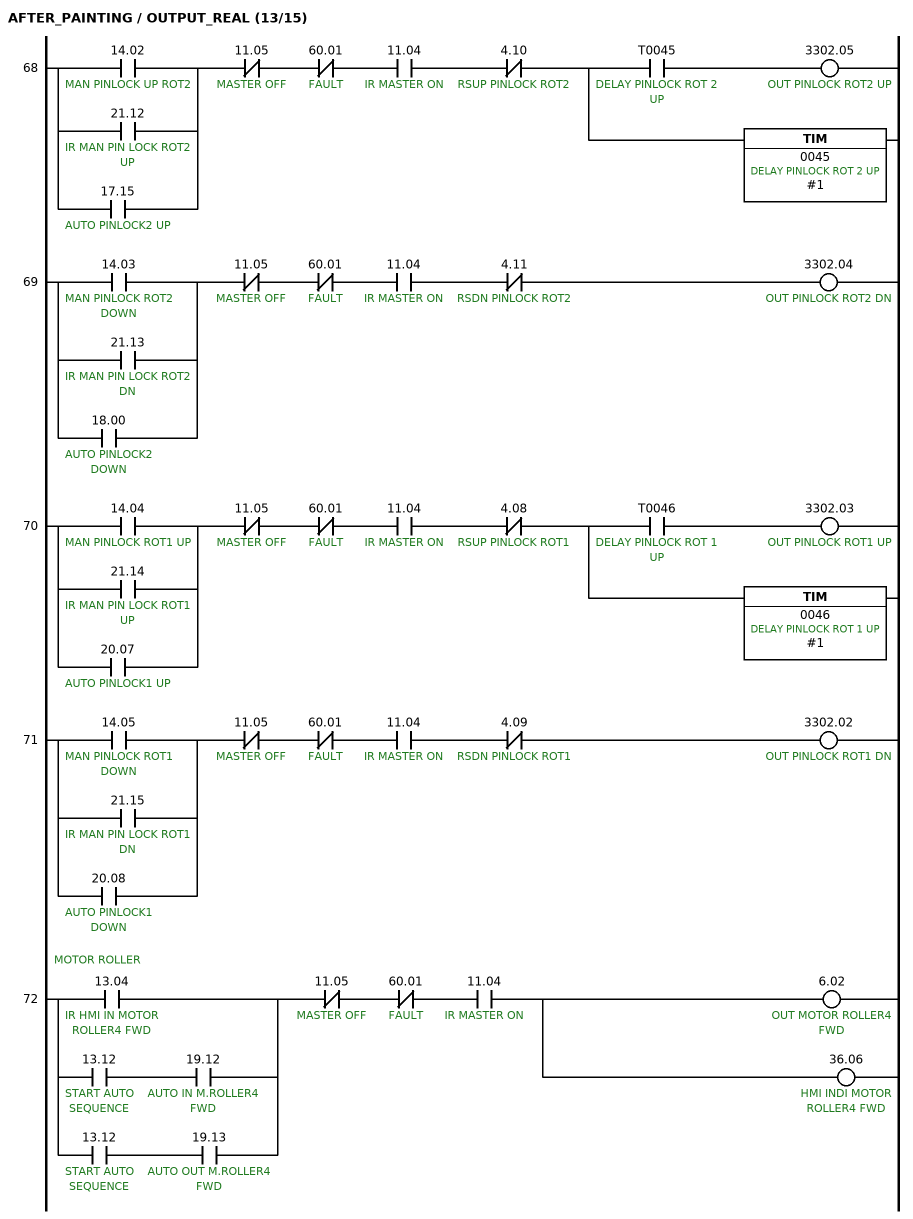
; [picture p24: AFTER_PAINTING / OUTPUT_REAL, rungs 68-72]
; rung 68
LD 14.02  ; MAN PINLOCK UP ROT2
OR 21.12  ; IR MAN PIN LOCK ROT2 UP
OR 17.15  ; AUTO PINLOCK2 UP
ANDNOT 11.05  ; MASTER OFF
ANDNOT 60.01  ; FAULT
AND 11.04  ; IR MASTER ON
ANDNOT 4.10  ; RSUP PINLOCK ROT2
OUT TR0
AND T0045  ; DELAY PINLOCK ROT 2 UP
OUT 3302.05  ; OUT PINLOCK ROT2 UP
LD TR0
TIM 0045 #1  ; DELAY PINLOCK ROT 2 UP
; rung 69
LD 14.03  ; MAN PINLOCK ROT2 DOWN
OR 21.13  ; IR MAN PIN LOCK ROT2 DN
OR 18.00  ; AUTO PINLOCK2 DOWN
ANDNOT 11.05  ; MASTER OFF
ANDNOT 60.01  ; FAULT
AND 11.04  ; IR MASTER ON
ANDNOT 4.11  ; RSDN PINLOCK ROT2
OUT 3302.04  ; OUT PINLOCK ROT2 DN
; rung 70
LD 14.04  ; MAN PINLOCK ROT1 UP
OR 21.14  ; IR MAN PIN LOCK ROT1 UP
OR 20.07  ; AUTO PINLOCK1 UP
ANDNOT 11.05  ; MASTER OFF
ANDNOT 60.01  ; FAULT
AND 11.04  ; IR MASTER ON
ANDNOT 4.08  ; RSUP PINLOCK ROT1
OUT TR0
AND T0046  ; DELAY PINLOCK ROT 1 UP
OUT 3302.03  ; OUT PINLOCK ROT1 UP
LD TR0
TIM 0046 #1  ; DELAY PINLOCK ROT 1 UP
; rung 71
LD 14.05  ; MAN PINLOCK ROT1 DOWN
OR 21.15  ; IR MAN PIN LOCK ROT1 DN
OR 20.08  ; AUTO PINLOCK1 DOWN
ANDNOT 11.05  ; MASTER OFF
ANDNOT 60.01  ; FAULT
AND 11.04  ; IR MASTER ON
ANDNOT 4.09  ; RSDN PINLOCK ROT1
OUT 3302.02  ; OUT PINLOCK ROT1 DN
; rung 72: MOTOR ROLLER
LD 13.04  ; IR HMI IN MOTOR ROLLER4 FWD
LD 13.12  ; START AUTO SEQUENCE
AND 19.12  ; AUTO IN M.ROLLER4 FWD
ORLD
LD 13.12  ; START AUTO SEQUENCE
AND 19.13  ; AUTO OUT M.ROLLER4 FWD
ORLD
ANDNOT 11.05  ; MASTER OFF
ANDNOT 60.01  ; FAULT
AND 11.04  ; IR MASTER ON
OUT 6.02  ; OUT MOTOR ROLLER4 FWD
OUT 36.06  ; HMI INDI MOTOR ROLLER4 FWD

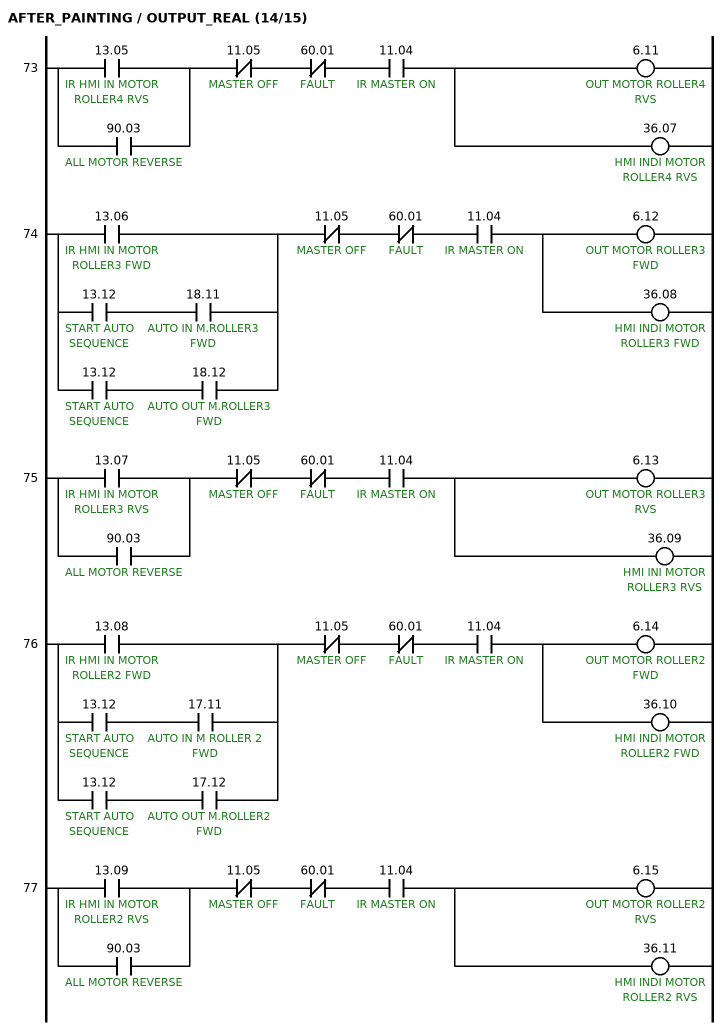
; rung 73
LD 13.05  ; IR HMI IN MOTOR ROLLER4 RVS
OR 90.03  ; ALL MOTOR REVERSE
ANDNOT 11.05  ; MASTER OFF
ANDNOT 60.01  ; FAULT
AND 11.04  ; IR MASTER ON
OUT 6.11  ; OUT MOTOR ROLLER4 RVS
OUT 36.07  ; HMI INDI MOTOR ROLLER4 RVS
; rung 74
LD 13.06  ; IR HMI IN MOTOR ROLLER3 FWD
LD 13.12  ; START AUTO SEQUENCE
AND 18.11  ; AUTO IN M.ROLLER3 FWD
ORLD
LD 13.12  ; START AUTO SEQUENCE
AND 18.12  ; AUTO OUT M.ROLLER3 FWD
ORLD
ANDNOT 11.05  ; MASTER OFF
ANDNOT 60.01  ; FAULT
AND 11.04  ; IR MASTER ON
OUT 6.12  ; OUT MOTOR ROLLER3 FWD
OUT 36.08  ; HMI INDI MOTOR ROLLER3 FWD
; rung 75
LD 13.07  ; IR HMI IN MOTOR ROLLER3 RVS
OR 90.03  ; ALL MOTOR REVERSE
ANDNOT 11.05  ; MASTER OFF
ANDNOT 60.01  ; FAULT
AND 11.04  ; IR MASTER ON
OUT 6.13  ; OUT MOTOR ROLLER3 RVS
OUT 36.09  ; HMI INI MOTOR ROLLER3 RVS
; rung 76
LD 13.08  ; IR HMI IN MOTOR ROLLER2 FWD
LD 13.12  ; START AUTO SEQUENCE
AND 17.11  ; AUTO IN M ROLLER 2 FWD
ORLD
LD 13.12  ; START AUTO SEQUENCE
AND 17.12  ; AUTO OUT M.ROLLER2 FWD
ORLD
ANDNOT 11.05  ; MASTER OFF
ANDNOT 60.01  ; FAULT
AND 11.04  ; IR MASTER ON
OUT 6.14  ; OUT MOTOR ROLLER2 FWD
OUT 36.10  ; HMI INDI MOTOR ROLLER2 FWD
; rung 77
LD 13.09  ; IR HMI IN MOTOR ROLLER2 RVS
OR 90.03  ; ALL MOTOR REVERSE
ANDNOT 11.05  ; MASTER OFF
ANDNOT 60.01  ; FAULT
AND 11.04  ; IR MASTER ON
OUT 6.15  ; OUT MOTOR ROLLER2 RVS
OUT 36.11  ; HMI INDI MOTOR ROLLER2 RVS

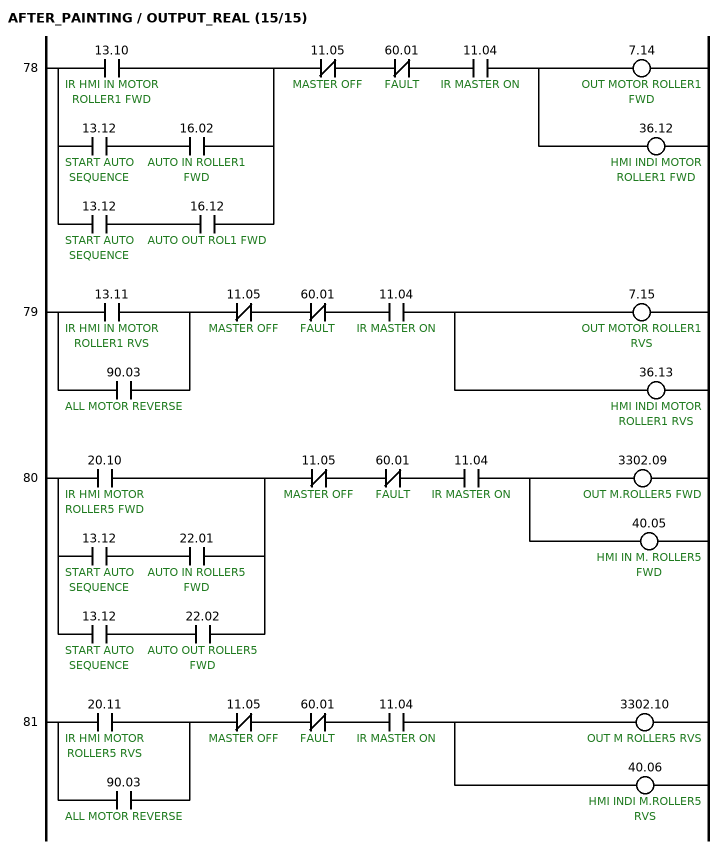
; rung 78
LD 13.10  ; IR HMI IN MOTOR ROLLER1 FWD
LD 13.12  ; START AUTO SEQUENCE
AND 16.02  ; AUTO IN ROLLER1 FWD
ORLD
LD 13.12  ; START AUTO SEQUENCE
AND 16.12  ; AUTO OUT ROL1 FWD
ORLD
ANDNOT 11.05  ; MASTER OFF
ANDNOT 60.01  ; FAULT
AND 11.04  ; IR MASTER ON
OUT 7.14  ; OUT MOTOR ROLLER1 FWD
OUT 36.12  ; HMI INDI MOTOR ROLLER1 FWD
; rung 79
LD 13.11  ; IR HMI IN MOTOR ROLLER1 RVS
OR 90.03  ; ALL MOTOR REVERSE
ANDNOT 11.05  ; MASTER OFF
ANDNOT 60.01  ; FAULT
AND 11.04  ; IR MASTER ON
OUT 7.15  ; OUT MOTOR ROLLER1 RVS
OUT 36.13  ; HMI INDI MOTOR ROLLER1 RVS
; rung 80
LD 20.10  ; IR HMI MOTOR ROLLER5 FWD
LD 13.12  ; START AUTO SEQUENCE
AND 22.01  ; AUTO IN ROLLER5 FWD
ORLD
LD 13.12  ; START AUTO SEQUENCE
AND 22.02  ; AUTO OUT ROLLER5 FWD
ORLD
ANDNOT 11.05  ; MASTER OFF
ANDNOT 60.01  ; FAULT
AND 11.04  ; IR MASTER ON
OUT 3302.09  ; OUT M.ROLLER5 FWD
OUT 40.05  ; HMI IN M. ROLLER5 FWD
; rung 81
LD 20.11  ; IR HMI MOTOR ROLLER5 RVS
OR 90.03  ; ALL MOTOR REVERSE
ANDNOT 11.05  ; MASTER OFF
ANDNOT 60.01  ; FAULT
AND 11.04  ; IR MASTER ON
OUT 3302.10  ; OUT M ROLLER5 RVS
OUT 40.06  ; HMI INDI M.ROLLER5 RVS

### Section MAIN

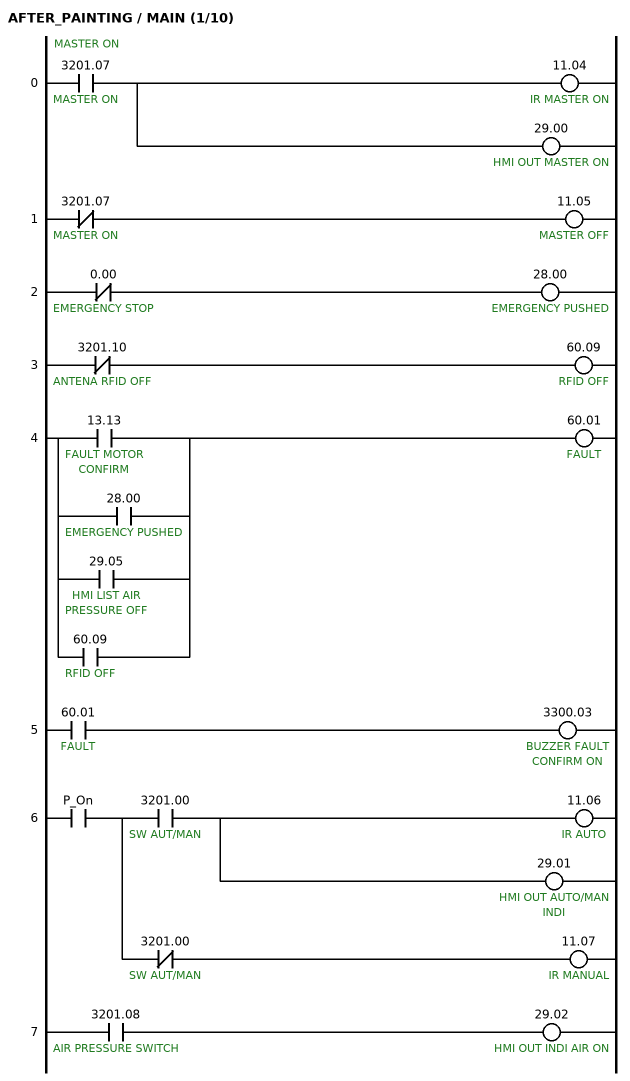
; rung 0: MASTER ON
LD 3201.07  ; MASTER ON
OUT 11.04  ; IR MASTER ON
OUT 29.00  ; HMI OUT MASTER ON
; rung 1
LDNOT 3201.07  ; MASTER ON
OUT 11.05  ; MASTER OFF
; rung 2
LDNOT 0.00  ; EMERGENCY STOP
OUT 28.00  ; EMERGENCY PUSHED
; rung 3
LDNOT 3201.10  ; ANTENA RFID OFF
OUT 60.09  ; RFID OFF
; rung 4
LD 13.13  ; FAULT MOTOR CONFIRM
OR 28.00  ; EMERGENCY PUSHED
OR 29.05  ; HMI LIST AIR PRESSURE OFF
OR 60.09  ; RFID OFF
OUT 60.01  ; FAULT
; rung 5
LD 60.01  ; FAULT
OUT 3300.03  ; BUZZER FAULT CONFIRM ON
; rung 6
LD P_On
OUT TR0
AND 3201.00  ; SW AUT/MAN
OUT 11.06  ; IR AUTO
OUT 29.01  ; HMI OUT AUTO/MAN INDI
LD TR0
ANDNOT 3201.00  ; SW AUT/MAN
OUT 11.07  ; IR MANUAL
; rung 7
LD 3201.08  ; AIR PRESSURE SWITCH
OUT 29.02  ; HMI OUT INDI AIR ON

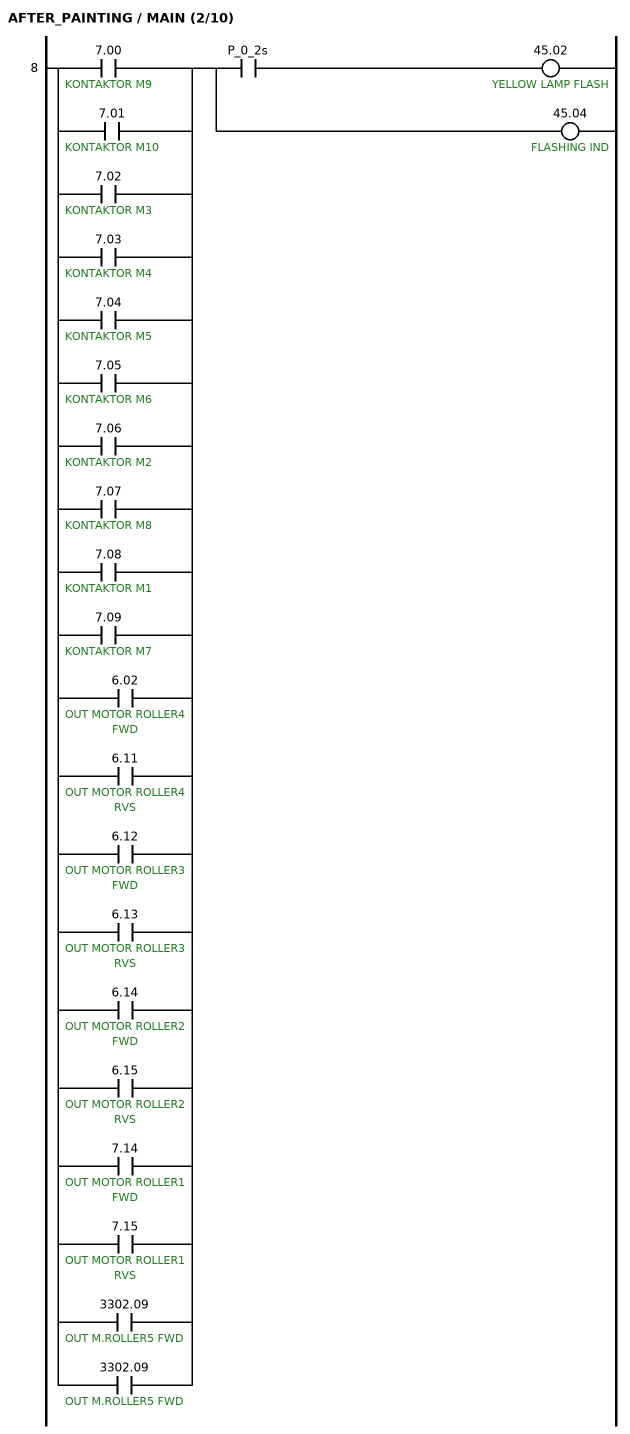
; rung 8
LD 7.00  ; KONTAKTOR M9
OR 7.01  ; KONTAKTOR M10
OR 7.02  ; KONTAKTOR M3
OR 7.03  ; KONTAKTOR M4
OR 7.04  ; KONTAKTOR M5
OR 7.05  ; KONTAKTOR M6
OR 7.06  ; KONTAKTOR M2
OR 7.07  ; KONTAKTOR M8
OR 7.08  ; KONTAKTOR M1
OR 7.09  ; KONTAKTOR M7
OR 6.02  ; OUT MOTOR ROLLER4 FWD
OR 6.11  ; OUT MOTOR ROLLER4 RVS
OR 6.12  ; OUT MOTOR ROLLER3 FWD
OR 6.13  ; OUT MOTOR ROLLER3 RVS
OR 6.14  ; OUT MOTOR ROLLER2 FWD
OR 6.15  ; OUT MOTOR ROLLER2 RVS
OR 7.14  ; OUT MOTOR ROLLER1 FWD
OR 7.15  ; OUT MOTOR ROLLER1 RVS
OR 3302.09  ; OUT M.ROLLER5 FWD
OR 3302.09  ; OUT M.ROLLER5 FWD
OUT TR0
AND P_0_2s
OUT 45.02  ; YELLOW LAMP FLASH
LD TR0
OUT 45.04  ; FLASHING IND

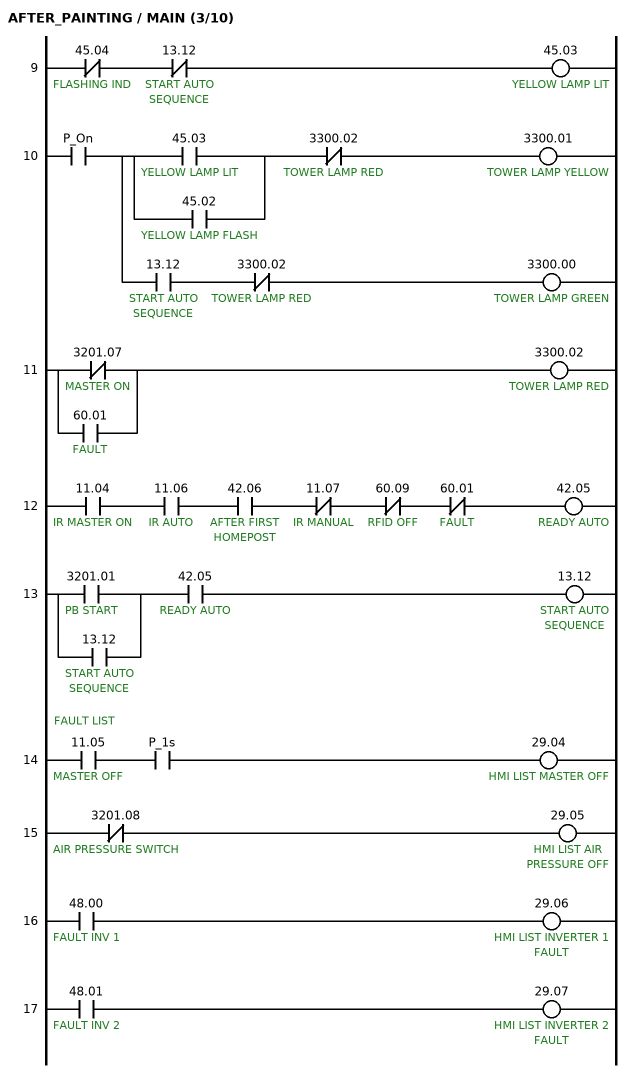
; rung 9
LDNOT 45.04  ; FLASHING IND
ANDNOT 13.12  ; START AUTO SEQUENCE
OUT 45.03  ; YELLOW LAMP LIT
; rung 10
LD P_On
OUT TR0
LD 45.03  ; YELLOW LAMP LIT
OR 45.02  ; YELLOW LAMP FLASH
ANDLD
ANDNOT 3300.02  ; TOWER LAMP RED
OUT 3300.01  ; TOWER LAMP YELLOW
LD TR0
AND 13.12  ; START AUTO SEQUENCE
ANDNOT 3300.02  ; TOWER LAMP RED
OUT 3300.00  ; TOWER LAMP GREEN
; rung 11
LDNOT 3201.07  ; MASTER ON
OR 60.01  ; FAULT
OUT 3300.02  ; TOWER LAMP RED
; rung 12
LD 11.04  ; IR MASTER ON
AND 11.06  ; IR AUTO
AND 42.06  ; AFTER FIRST HOMEPOST
ANDNOT 11.07  ; IR MANUAL
ANDNOT 60.09  ; RFID OFF
ANDNOT 60.01  ; FAULT
OUT 42.05  ; READY AUTO
; rung 13
LD 3201.01  ; PB START
OR 13.12  ; START AUTO SEQUENCE
AND 42.05  ; READY AUTO
OUT 13.12  ; START AUTO SEQUENCE
; rung 14: FAULT LIST
LD 11.05  ; MASTER OFF
AND P_1s
OUT 29.04  ; HMI LIST MASTER OFF
; rung 15
LDNOT 3201.08  ; AIR PRESSURE SWITCH
OUT 29.05  ; HMI LIST AIR PRESSURE OFF
; rung 16
LD 48.00  ; FAULT INV 1
OUT 29.06  ; HMI LIST INVERTER 1 FAULT
; rung 17
LD 48.01  ; FAULT INV 2
OUT 29.07  ; HMI LIST INVERTER 2 FAULT

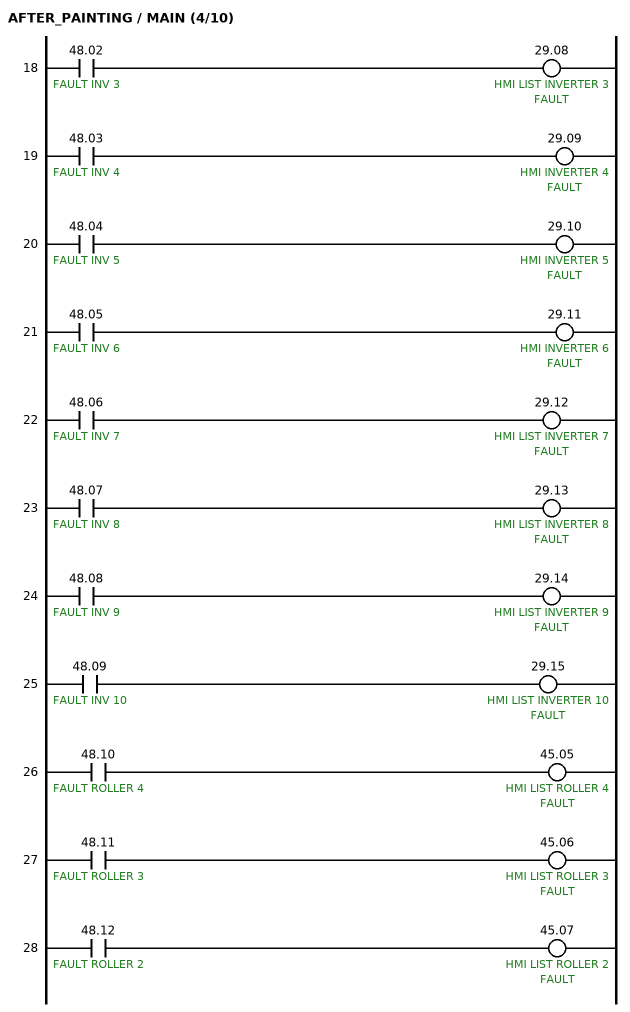
; rung 18
LD 48.02  ; FAULT INV 3
OUT 29.08  ; HMI LIST INVERTER 3 FAULT
; rung 19
LD 48.03  ; FAULT INV 4
OUT 29.09  ; HMI INVERTER 4 FAULT
; rung 20
LD 48.04  ; FAULT INV 5
OUT 29.10  ; HMI INVERTER 5 FAULT
; rung 21
LD 48.05  ; FAULT INV 6
OUT 29.11  ; HMI INVERTER 6 FAULT
; rung 22
LD 48.06  ; FAULT INV 7
OUT 29.12  ; HMI LIST INVERTER 7 FAULT
; rung 23
LD 48.07  ; FAULT INV 8
OUT 29.13  ; HMI LIST INVERTER 8 FAULT
; rung 24
LD 48.08  ; FAULT INV 9
OUT 29.14  ; HMI LIST INVERTER 9 FAULT
; rung 25
LD 48.09  ; FAULT INV 10
OUT 29.15  ; HMI LIST INVERTER 10 FAULT
; rung 26
LD 48.10  ; FAULT ROLLER 4
OUT 45.05  ; HMI LIST ROLLER 4 FAULT
; rung 27
LD 48.11  ; FAULT ROLLER 3
OUT 45.06  ; HMI LIST ROLLER 3 FAULT
; rung 28
LD 48.12  ; FAULT ROLLER 2
OUT 45.07  ; HMI LIST ROLLER 2 FAULT

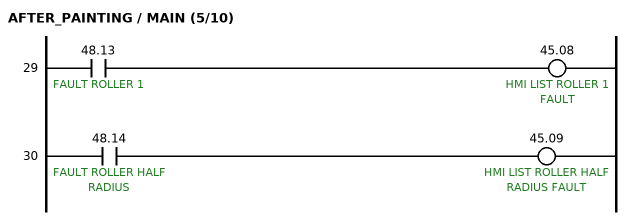
; rung 29
LD 48.13  ; FAULT ROLLER 1
OUT 45.08  ; HMI LIST ROLLER 1 FAULT
; rung 30
LD 48.14  ; FAULT ROLLER HALF RADIUS
OUT 45.09  ; HMI LIST ROLLER HALF RADIUS FAULT

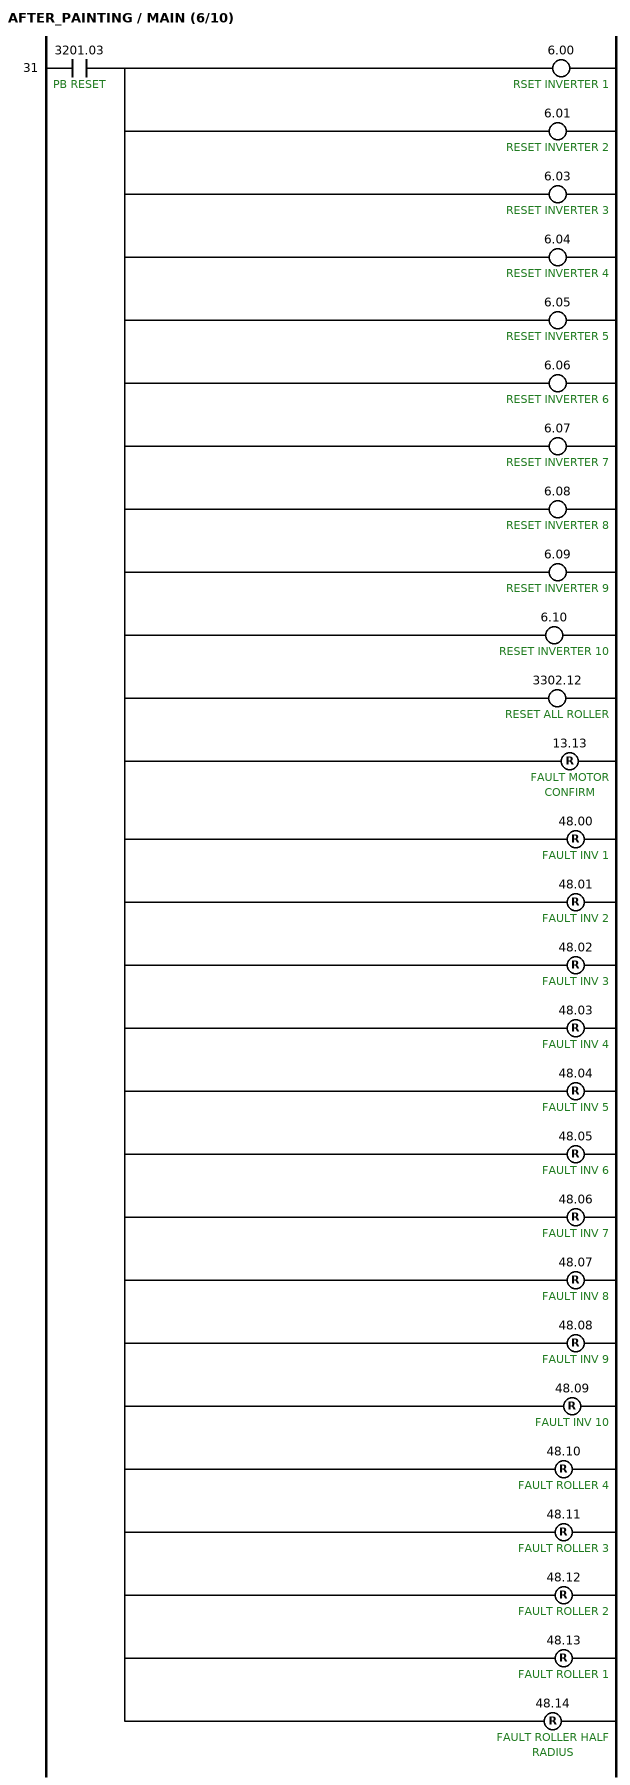
; rung 31
LD 3201.03  ; PB RESET
OUT 6.00  ; RSET INVERTER 1
OUT 6.01  ; RESET INVERTER 2
OUT 6.03  ; RESET INVERTER 3
OUT 6.04  ; RESET INVERTER 4
OUT 6.05  ; RESET INVERTER 5
OUT 6.06  ; RESET INVERTER 6
OUT 6.07  ; RESET INVERTER 7
OUT 6.08  ; RESET INVERTER 8
OUT 6.09  ; RESET INVERTER 9
OUT 6.10  ; RESET INVERTER 10
OUT 3302.12  ; RESET ALL ROLLER
RSET 13.13  ; FAULT MOTOR CONFIRM
RSET 48.00  ; FAULT INV 1
RSET 48.01  ; FAULT INV 2
RSET 48.02  ; FAULT INV 3
RSET 48.03  ; FAULT INV 4
RSET 48.04  ; FAULT INV 5
RSET 48.05  ; FAULT INV 6
RSET 48.06  ; FAULT INV 7
RSET 48.07  ; FAULT INV 8
RSET 48.08  ; FAULT INV 9
RSET 48.09  ; FAULT INV 10
RSET 48.10  ; FAULT ROLLER 4
RSET 48.11  ; FAULT ROLLER 3
RSET 48.12  ; FAULT ROLLER 2
RSET 48.13  ; FAULT ROLLER 1
RSET 48.14  ; FAULT ROLLER HALF RADIUS

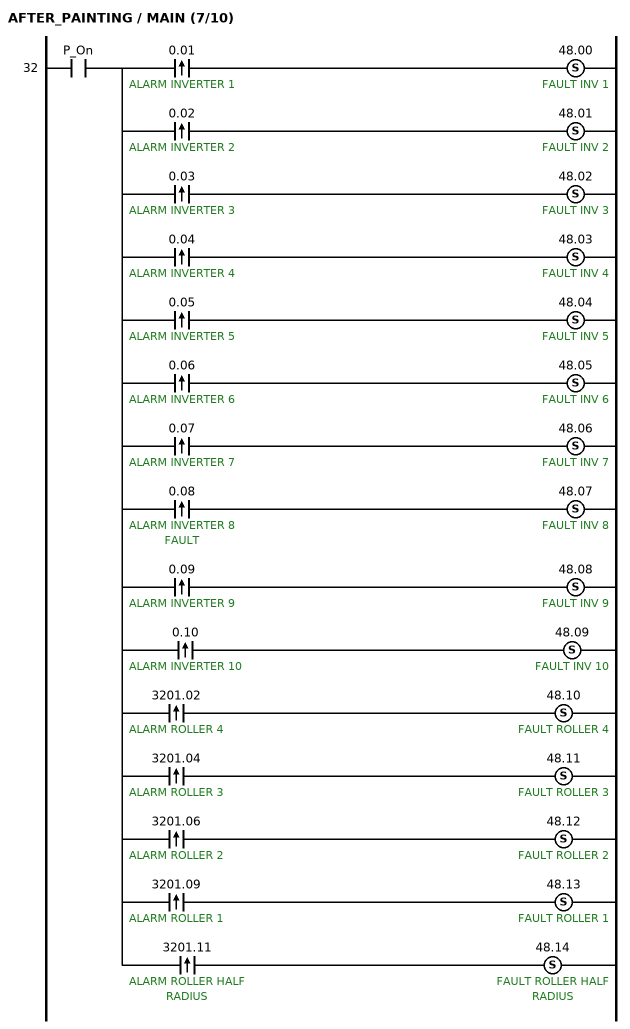
; rung 32
LD P_On
OUT TR0
@AND 0.01  ; ALARM INVERTER 1
SET 48.00  ; FAULT INV 1
LD TR0
@AND 0.02  ; ALARM INVERTER 2
SET 48.01  ; FAULT INV 2
LD TR0
@AND 0.03  ; ALARM INVERTER 3
SET 48.02  ; FAULT INV 3
LD TR0
@AND 0.04  ; ALARM INVERTER 4
SET 48.03  ; FAULT INV 4
LD TR0
@AND 0.05  ; ALARM INVERTER 5
SET 48.04  ; FAULT INV 5
LD TR0
@AND 0.06  ; ALARM INVERTER 6
SET 48.05  ; FAULT INV 6
LD TR0
@AND 0.07  ; ALARM INVERTER 7
SET 48.06  ; FAULT INV 7
LD TR0
@AND 0.08  ; ALARM INVERTER 8 FAULT
SET 48.07  ; FAULT INV 8
LD TR0
@AND 0.09  ; ALARM INVERTER 9
SET 48.08  ; FAULT INV 9
LD TR0
@AND 0.10  ; ALARM INVERTER 10
SET 48.09  ; FAULT INV 10
LD TR0
@AND 3201.02  ; ALARM ROLLER 4
SET 48.10  ; FAULT ROLLER 4
LD TR0
@AND 3201.04  ; ALARM ROLLER 3
SET 48.11  ; FAULT ROLLER 3
LD TR0
@AND 3201.06  ; ALARM ROLLER 2
SET 48.12  ; FAULT ROLLER 2
LD TR0
@AND 3201.09  ; ALARM ROLLER 1
SET 48.13  ; FAULT ROLLER 1
LD TR0
@AND 3201.11  ; ALARM ROLLER HALF RADIUS
SET 48.14  ; FAULT ROLLER HALF RADIUS

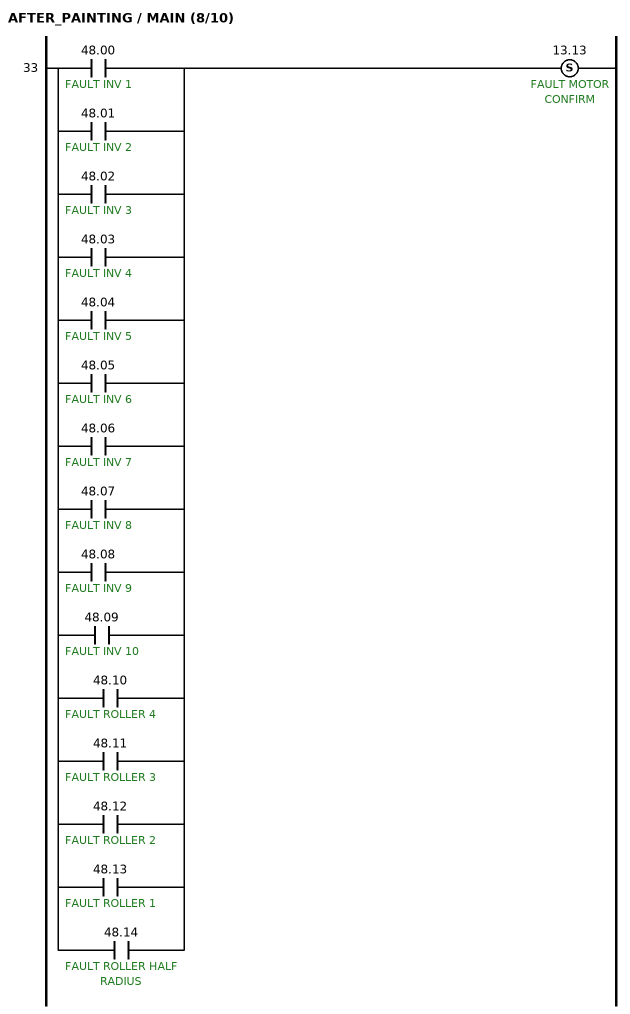
; rung 33
LD 48.00  ; FAULT INV 1
OR 48.01  ; FAULT INV 2
OR 48.02  ; FAULT INV 3
OR 48.03  ; FAULT INV 4
OR 48.04  ; FAULT INV 5
OR 48.05  ; FAULT INV 6
OR 48.06  ; FAULT INV 7
OR 48.07  ; FAULT INV 8
OR 48.08  ; FAULT INV 9
OR 48.09  ; FAULT INV 10
OR 48.10  ; FAULT ROLLER 4
OR 48.11  ; FAULT ROLLER 3
OR 48.12  ; FAULT ROLLER 2
OR 48.13  ; FAULT ROLLER 1
OR 48.14  ; FAULT ROLLER HALF RADIUS
SET 13.13  ; FAULT MOTOR CONFIRM

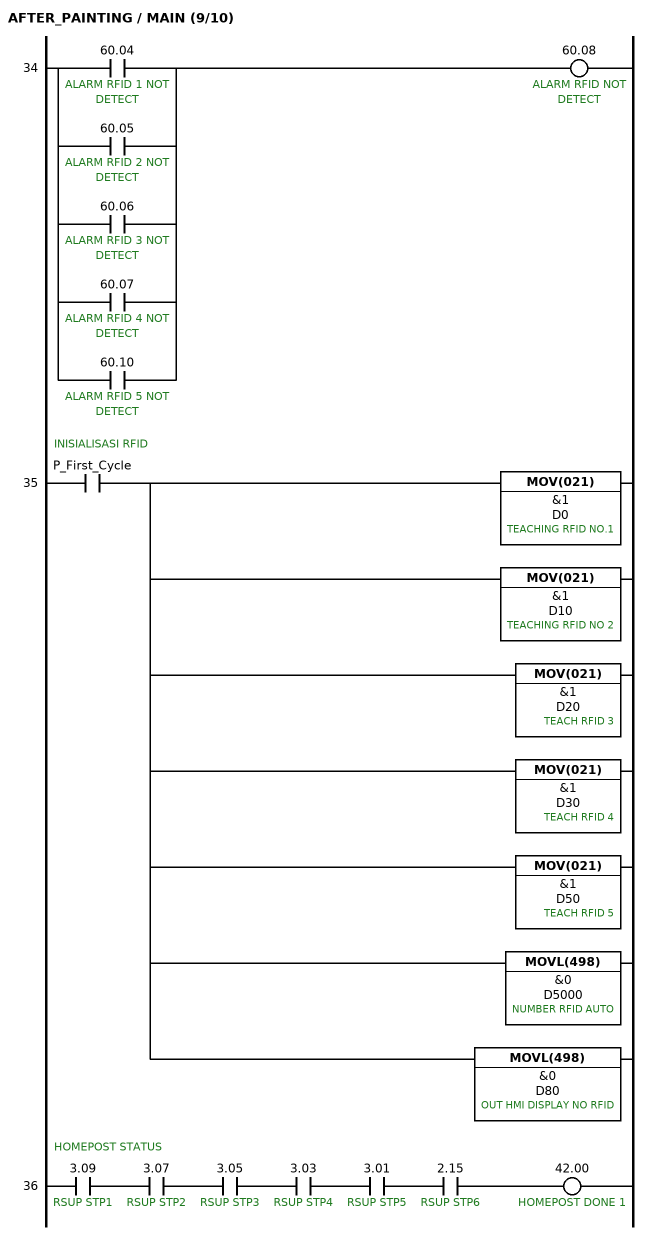
; rung 34
LD 60.04  ; ALARM RFID 1 NOT DETECT
OR 60.05  ; ALARM RFID 2 NOT DETECT
OR 60.06  ; ALARM RFID 3 NOT DETECT
OR 60.07  ; ALARM RFID 4 NOT DETECT
OR 60.10  ; ALARM RFID 5 NOT DETECT
OUT 60.08  ; ALARM RFID NOT DETECT
; rung 35: INISIALISASI RFID
LD P_First_Cycle
MOV(021) &1 D0  ; TEACHING RFID NO.1
MOV(021) &1 D10  ; TEACHING RFID NO 2
MOV(021) &1 D20  ; TEACH RFID 3
MOV(021) &1 D30  ; TEACH RFID 4
MOV(021) &1 D50  ; TEACH RFID 5
MOVL(498) &0 D5000  ; NUMBER RFID AUTO
MOVL(498) &0 D80  ; OUT HMI DISPLAY NO RFID
; rung 36: HOMEPOST STATUS
LD 3.09  ; RSUP STP1
AND 3.07  ; RSUP STP2
AND 3.05  ; RSUP STP3
AND 3.03  ; RSUP STP4
AND 3.01  ; RSUP STP5
AND 2.15  ; RSUP STP6
OUT 42.00  ; HOMEPOST DONE 1

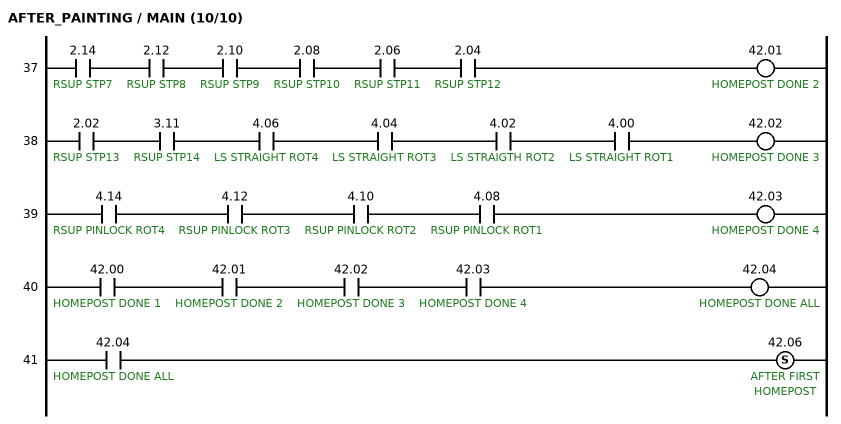
; rung 37
LD 2.14  ; RSUP STP7
AND 2.12  ; RSUP STP8
AND 2.10  ; RSUP STP9
AND 2.08  ; RSUP STP10
AND 2.06  ; RSUP STP11
AND 2.04  ; RSUP STP12
OUT 42.01  ; HOMEPOST DONE 2
; rung 38
LD 2.02  ; RSUP STP13
AND 3.11  ; RSUP STP14
AND 4.06  ; LS STRAIGHT ROT4
AND 4.04  ; LS STRAIGHT ROT3
AND 4.02  ; LS STRAIGTH ROT2
AND 4.00  ; LS STRAIGHT ROT1
OUT 42.02  ; HOMEPOST DONE 3
; rung 39
LD 4.14  ; RSUP PINLOCK ROT4
AND 4.12  ; RSUP PINLOCK ROT3
AND 4.10  ; RSUP PINLOCK ROT2
AND 4.08  ; RSUP PINLOCK ROT1
OUT 42.03  ; HOMEPOST DONE 4
; rung 40
LD 42.00  ; HOMEPOST DONE 1
AND 42.01  ; HOMEPOST DONE 2
AND 42.02  ; HOMEPOST DONE 3
AND 42.03  ; HOMEPOST DONE 4
OUT 42.04  ; HOMEPOST DONE ALL
; rung 41
LD 42.04  ; HOMEPOST DONE ALL
SET 42.06  ; AFTER FIRST HOMEPOST

### Section INPUT

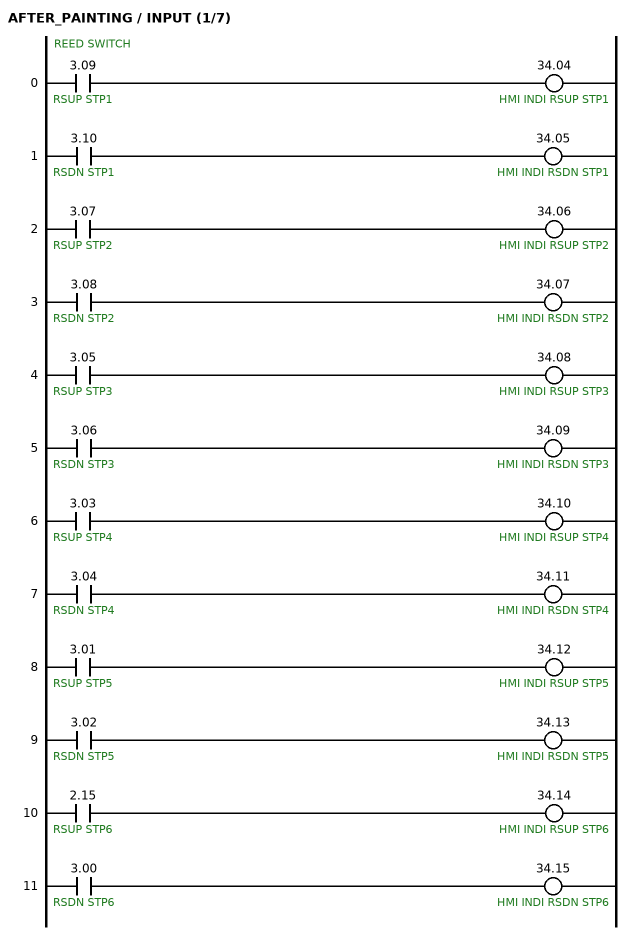
; rung 0: REED SWITCH
LD 3.09  ; RSUP STP1
OUT 34.04  ; HMI INDI RSUP STP1
; rung 1
LD 3.10  ; RSDN STP1
OUT 34.05  ; HMI INDI RSDN STP1
; rung 2
LD 3.07  ; RSUP STP2
OUT 34.06  ; HMI INDI RSUP STP2
; rung 3
LD 3.08  ; RSDN STP2
OUT 34.07  ; HMI INDI RSDN STP2
; rung 4
LD 3.05  ; RSUP STP3
OUT 34.08  ; HMI INDI RSUP STP3
; rung 5
LD 3.06  ; RSDN STP3
OUT 34.09  ; HMI INDI RSDN STP3
; rung 6
LD 3.03  ; RSUP STP4
OUT 34.10  ; HMI INDI RSUP STP4
; rung 7
LD 3.04  ; RSDN STP4
OUT 34.11  ; HMI INDI RSDN STP4
; rung 8
LD 3.01  ; RSUP STP5
OUT 34.12  ; HMI INDI RSUP STP5
; rung 9
LD 3.02  ; RSDN STP5
OUT 34.13  ; HMI INDI RSDN STP5
; rung 10
LD 2.15  ; RSUP STP6
OUT 34.14  ; HMI INDI RSUP STP6
; rung 11
LD 3.00  ; RSDN STP6
OUT 34.15  ; HMI INDI RSDN STP6

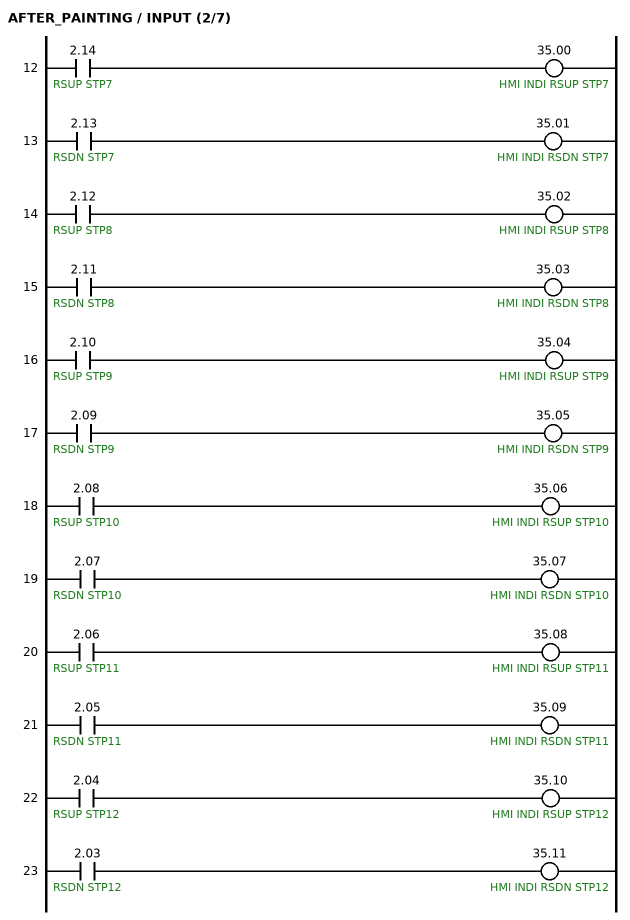
; rung 12
LD 2.14  ; RSUP STP7
OUT 35.00  ; HMI INDI RSUP STP7
; rung 13
LD 2.13  ; RSDN STP7
OUT 35.01  ; HMI INDI RSDN STP7
; rung 14
LD 2.12  ; RSUP STP8
OUT 35.02  ; HMI INDI RSUP STP8
; rung 15
LD 2.11  ; RSDN STP8
OUT 35.03  ; HMI INDI RSDN STP8
; rung 16
LD 2.10  ; RSUP STP9
OUT 35.04  ; HMI INDI RSUP STP9
; rung 17
LD 2.09  ; RSDN STP9
OUT 35.05  ; HMI INDI RSDN STP9
; rung 18
LD 2.08  ; RSUP STP10
OUT 35.06  ; HMI INDI RSUP STP10
; rung 19
LD 2.07  ; RSDN STP10
OUT 35.07  ; HMI INDI RSDN STP10
; rung 20
LD 2.06  ; RSUP STP11
OUT 35.08  ; HMI INDI RSUP STP11
; rung 21
LD 2.05  ; RSDN STP11
OUT 35.09  ; HMI INDI RSDN STP11
; rung 22
LD 2.04  ; RSUP STP12
OUT 35.10  ; HMI INDI RSUP STP12
; rung 23
LD 2.03  ; RSDN STP12
OUT 35.11  ; HMI INDI RSDN STP12

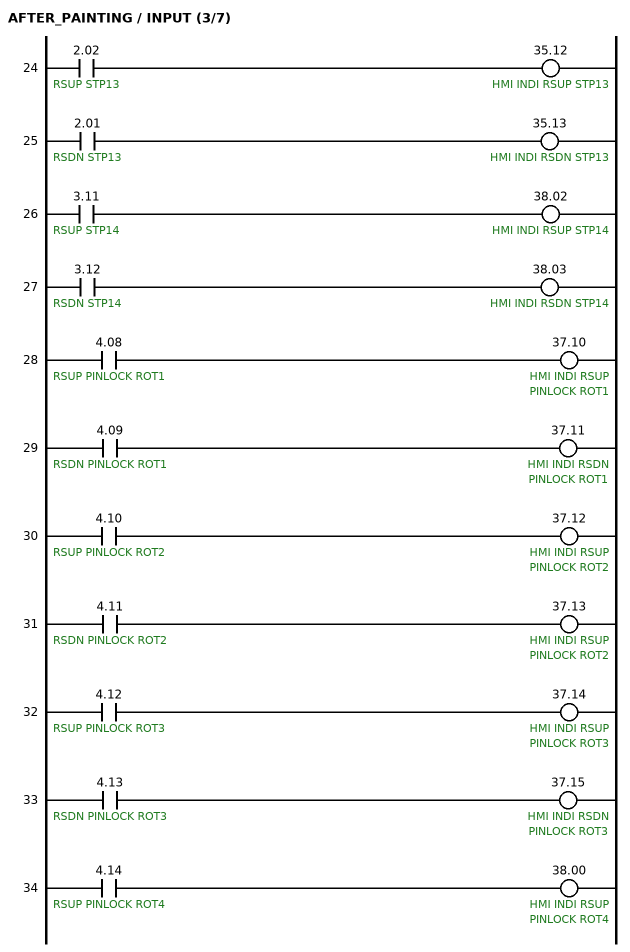
; rung 24
LD 2.02  ; RSUP STP13
OUT 35.12  ; HMI INDI RSUP STP13
; rung 25
LD 2.01  ; RSDN STP13
OUT 35.13  ; HMI INDI RSDN STP13
; rung 26
LD 3.11  ; RSUP STP14
OUT 38.02  ; HMI INDI RSUP STP14
; rung 27
LD 3.12  ; RSDN STP14
OUT 38.03  ; HMI INDI RSDN STP14
; rung 28
LD 4.08  ; RSUP PINLOCK ROT1
OUT 37.10  ; HMI INDI RSUP PINLOCK ROT1
; rung 29
LD 4.09  ; RSDN PINLOCK ROT1
OUT 37.11  ; HMI INDI RSDN PINLOCK ROT1
; rung 30
LD 4.10  ; RSUP PINLOCK ROT2
OUT 37.12  ; HMI INDI RSUP PINLOCK ROT2
; rung 31
LD 4.11  ; RSDN PINLOCK ROT2
OUT 37.13  ; HMI INDI RSUP PINLOCK ROT2
; rung 32
LD 4.12  ; RSUP PINLOCK ROT3
OUT 37.14  ; HMI INDI RSUP PINLOCK ROT3
; rung 33
LD 4.13  ; RSDN PINLOCK ROT3
OUT 37.15  ; HMI INDI RSDN PINLOCK ROT3
; rung 34
LD 4.14  ; RSUP PINLOCK ROT4
OUT 38.00  ; HMI INDI RSUP PINLOCK ROT4

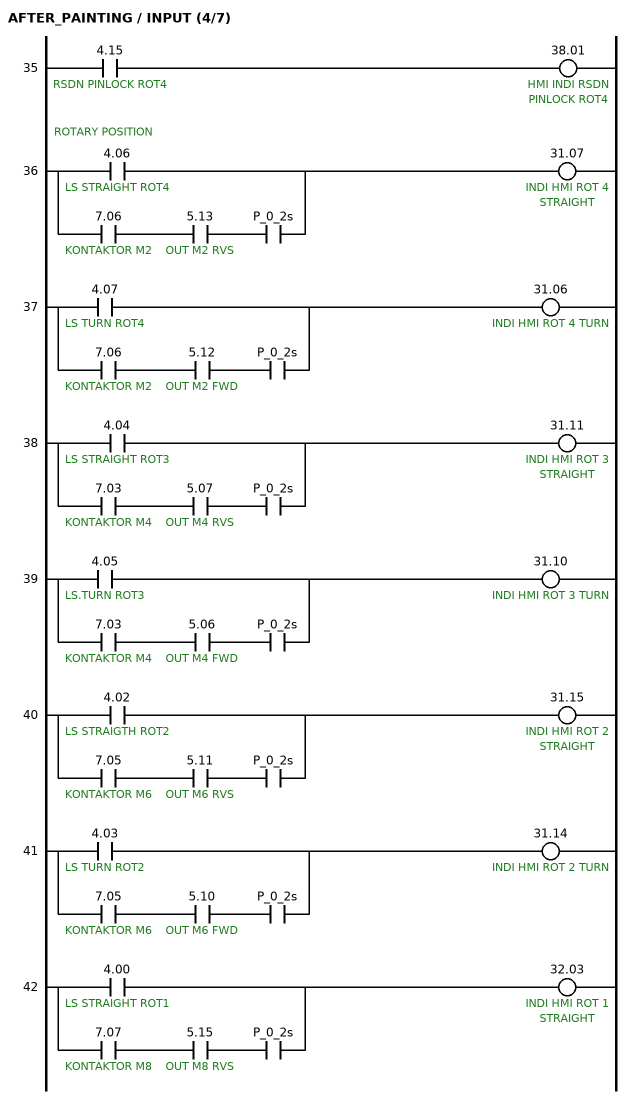
; rung 35
LD 4.15  ; RSDN PINLOCK ROT4
OUT 38.01  ; HMI INDI RSDN PINLOCK ROT4
; rung 36: ROTARY POSITION
LD 4.06  ; LS STRAIGHT ROT4
LD 7.06  ; KONTAKTOR M2
AND 5.13  ; OUT M2 RVS
AND P_0_2s
ORLD
OUT 31.07  ; INDI HMI ROT 4 STRAIGHT
; rung 37
LD 4.07  ; LS TURN ROT4
LD 7.06  ; KONTAKTOR M2
AND 5.12  ; OUT M2 FWD
AND P_0_2s
ORLD
OUT 31.06  ; INDI HMI ROT 4 TURN
; rung 38
LD 4.04  ; LS STRAIGHT ROT3
LD 7.03  ; KONTAKTOR M4
AND 5.07  ; OUT M4 RVS
AND P_0_2s
ORLD
OUT 31.11  ; INDI HMI ROT 3 STRAIGHT
; rung 39
LD 4.05  ; LS.TURN ROT3
LD 7.03  ; KONTAKTOR M4
AND 5.06  ; OUT M4 FWD
AND P_0_2s
ORLD
OUT 31.10  ; INDI HMI ROT 3 TURN
; rung 40
LD 4.02  ; LS STRAIGTH ROT2
LD 7.05  ; KONTAKTOR M6
AND 5.11  ; OUT M6 RVS
AND P_0_2s
ORLD
OUT 31.15  ; INDI HMI ROT 2 STRAIGHT
; rung 41
LD 4.03  ; LS TURN ROT2
LD 7.05  ; KONTAKTOR M6
AND 5.10  ; OUT M6 FWD
AND P_0_2s
ORLD
OUT 31.14  ; INDI HMI ROT 2 TURN
; rung 42
LD 4.00  ; LS STRAIGHT ROT1
LD 7.07  ; KONTAKTOR M8
AND 5.15  ; OUT M8 RVS
AND P_0_2s
ORLD
OUT 32.03  ; INDI HMI ROT 1 STRAIGHT

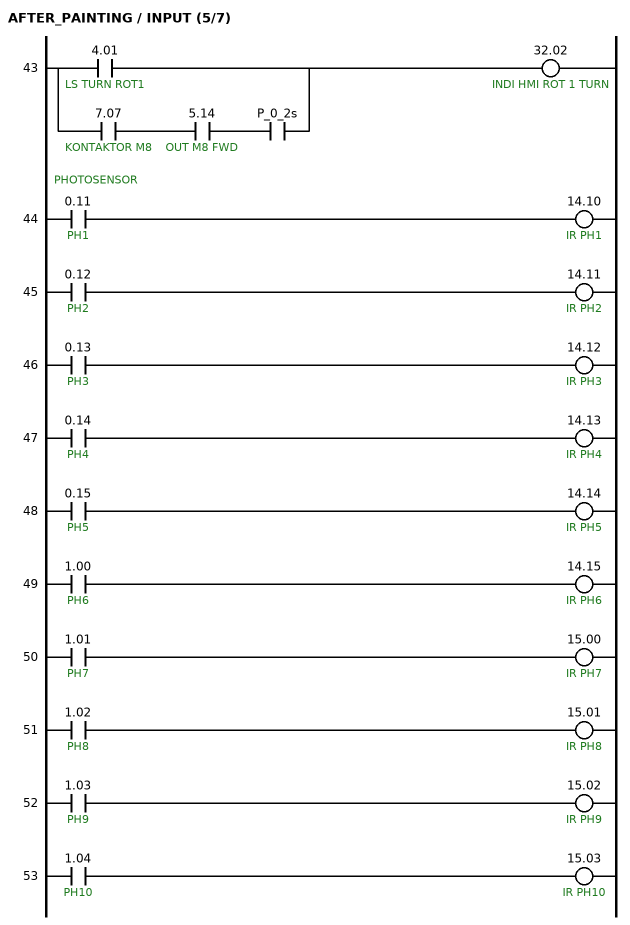
; rung 43
LD 4.01  ; LS TURN ROT1
LD 7.07  ; KONTAKTOR M8
AND 5.14  ; OUT M8 FWD
AND P_0_2s
ORLD
OUT 32.02  ; INDI HMI ROT 1 TURN
; rung 44: PHOTOSENSOR
LD 0.11  ; PH1
OUT 14.10  ; IR PH1
; rung 45
LD 0.12  ; PH2
OUT 14.11  ; IR PH2
; rung 46
LD 0.13  ; PH3
OUT 14.12  ; IR PH3
; rung 47
LD 0.14  ; PH4
OUT 14.13  ; IR PH4
; rung 48
LD 0.15  ; PH5
OUT 14.14  ; IR PH5
; rung 49
LD 1.00  ; PH6
OUT 14.15  ; IR PH6
; rung 50
LD 1.01  ; PH7
OUT 15.00  ; IR PH7
; rung 51
LD 1.02  ; PH8
OUT 15.01  ; IR PH8
; rung 52
LD 1.03  ; PH9
OUT 15.02  ; IR PH9
; rung 53
LD 1.04  ; PH10
OUT 15.03  ; IR PH10

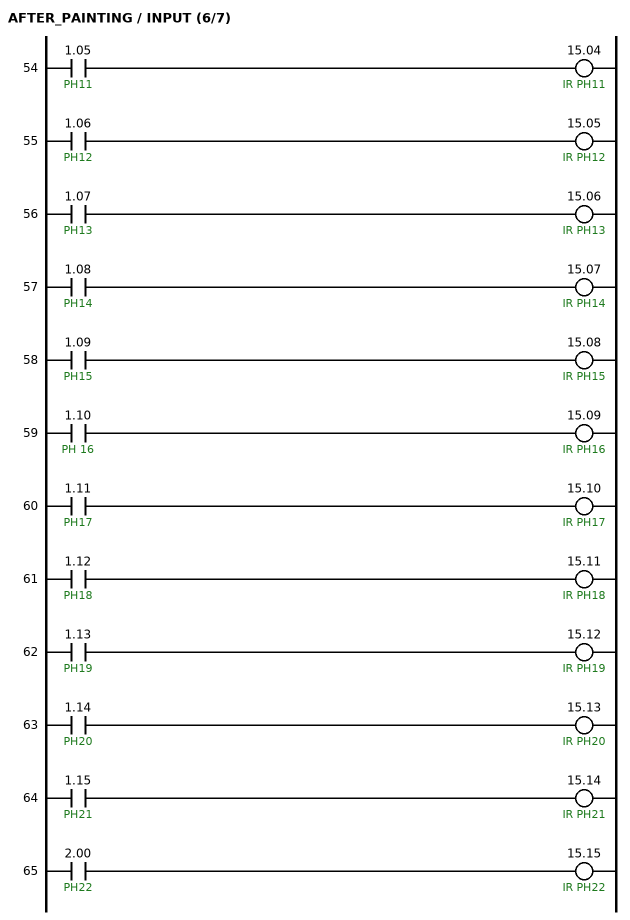
; rung 54
LD 1.05  ; PH11
OUT 15.04  ; IR PH11
; rung 55
LD 1.06  ; PH12
OUT 15.05  ; IR PH12
; rung 56
LD 1.07  ; PH13
OUT 15.06  ; IR PH13
; rung 57
LD 1.08  ; PH14
OUT 15.07  ; IR PH14
; rung 58
LD 1.09  ; PH15
OUT 15.08  ; IR PH15
; rung 59
LD 1.10  ; PH 16
OUT 15.09  ; IR PH16
; rung 60
LD 1.11  ; PH17
OUT 15.10  ; IR PH17
; rung 61
LD 1.12  ; PH18
OUT 15.11  ; IR PH18
; rung 62
LD 1.13  ; PH19
OUT 15.12  ; IR PH19
; rung 63
LD 1.14  ; PH20
OUT 15.13  ; IR PH20
; rung 64
LD 1.15  ; PH21
OUT 15.14  ; IR PH21
; rung 65
LD 2.00  ; PH22
OUT 15.15  ; IR PH22

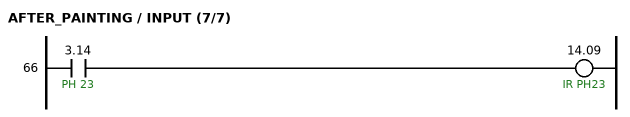
; rung 66
LD 3.14  ; PH 23
OUT 14.09  ; IR PH23

### Section SEQ_TOMBOL_HMI

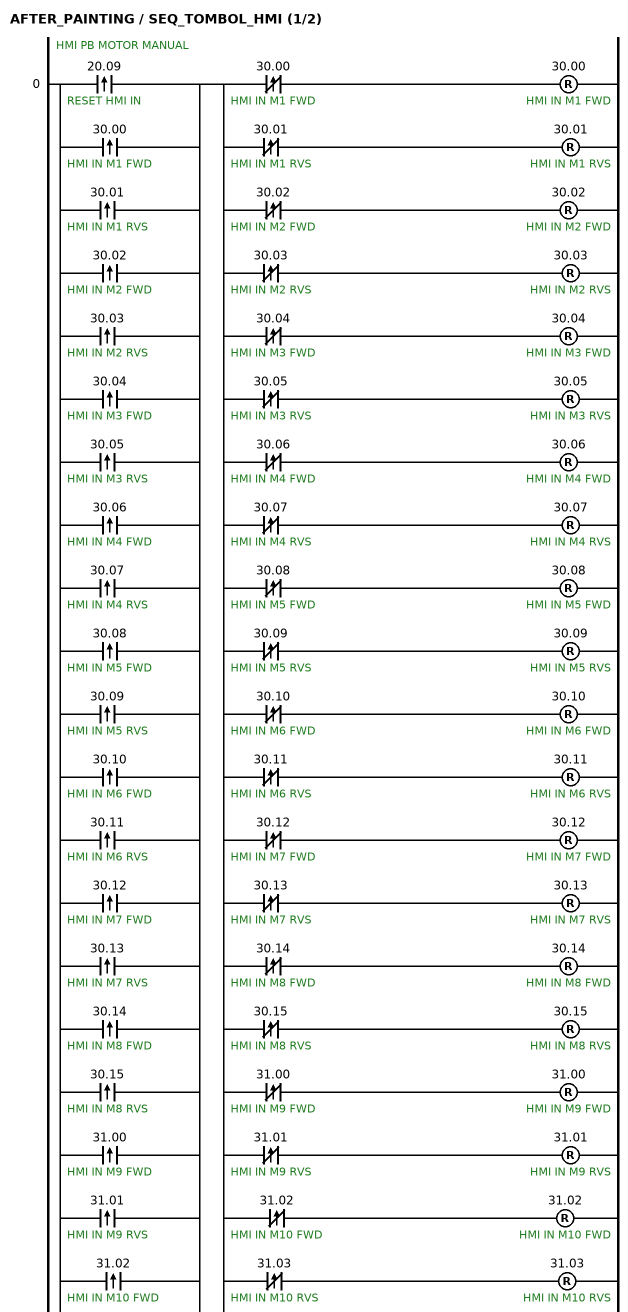

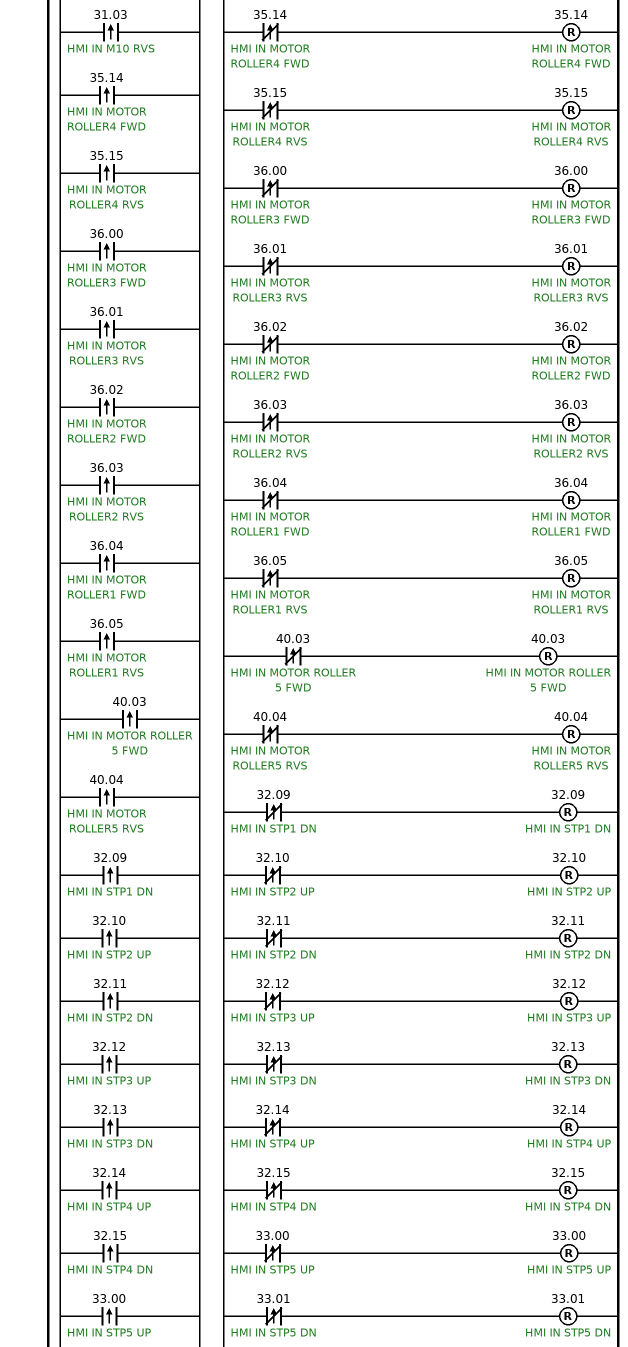

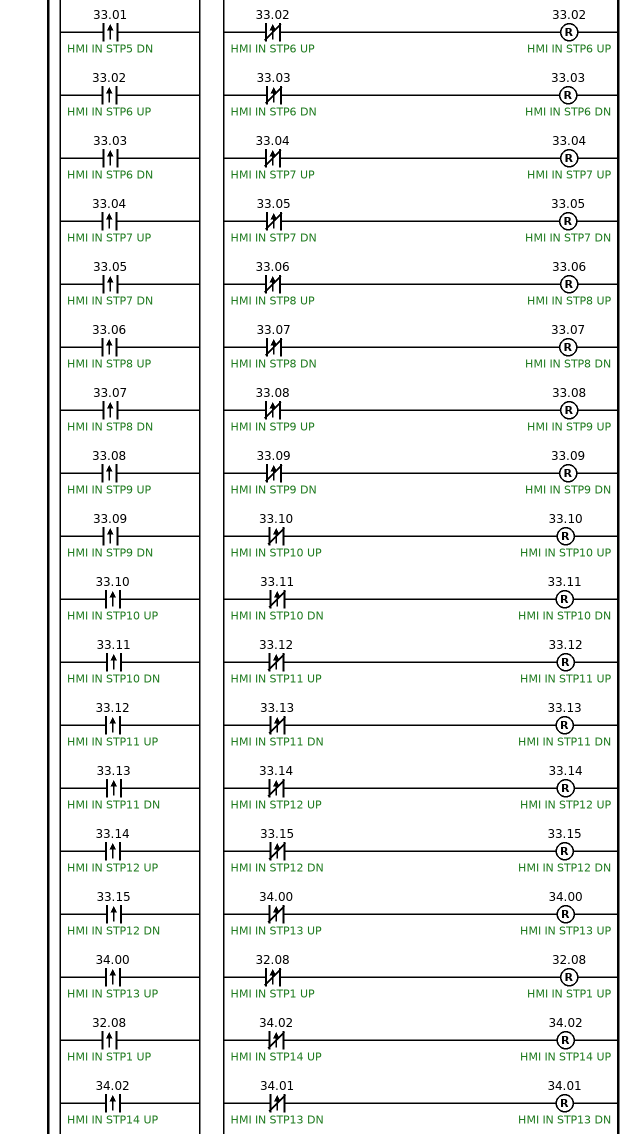

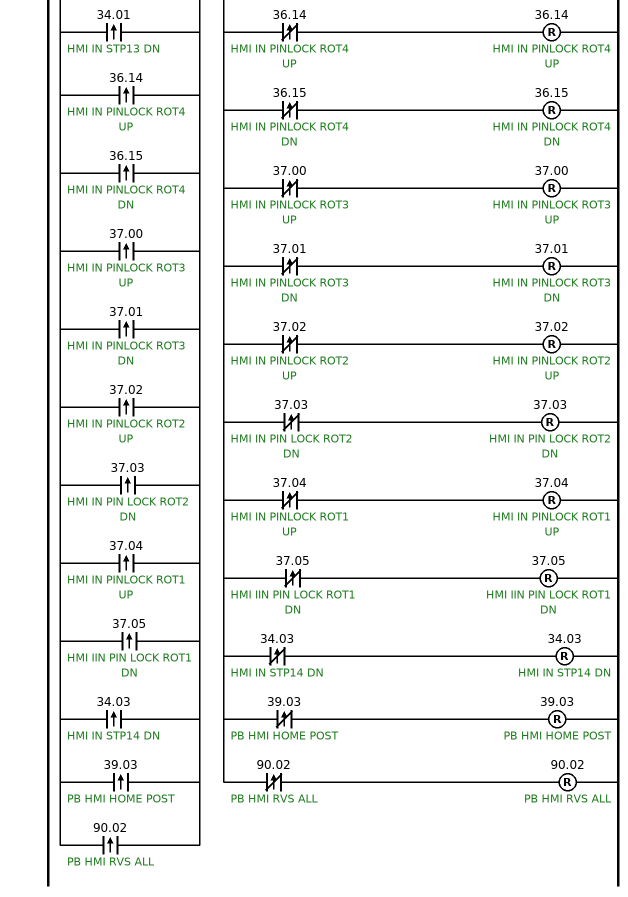
; rung 0: HMI PB MOTOR MANUAL
@LD 20.09  ; RESET HMI IN
@OR 30.00  ; HMI IN M1 FWD
@OR 30.01  ; HMI IN M1 RVS
@OR 30.02  ; HMI IN M2 FWD
@OR 30.03  ; HMI IN M2 RVS
@OR 30.04  ; HMI IN M3 FWD
@OR 30.05  ; HMI IN M3 RVS
@OR 30.06  ; HMI IN M4 FWD
@OR 30.07  ; HMI IN M4 RVS
@OR 30.08  ; HMI IN M5 FWD
@OR 30.09  ; HMI IN M5 RVS
@OR 30.10  ; HMI IN M6 FWD
@OR 30.11  ; HMI IN M6 RVS
@OR 30.12  ; HMI IN M7 FWD
@OR 30.13  ; HMI IN M7 RVS
@OR 30.14  ; HMI IN M8 FWD
@OR 30.15  ; HMI IN M8 RVS
@OR 31.00  ; HMI IN M9 FWD
@OR 31.01  ; HMI IN M9 RVS
@OR 31.02  ; HMI IN M10 FWD
@OR 31.03  ; HMI IN M10 RVS
@OR 35.14  ; HMI IN MOTOR ROLLER4 FWD
@OR 35.15  ; HMI IN MOTOR ROLLER4 RVS
@OR 36.00  ; HMI IN MOTOR ROLLER3 FWD
@OR 36.01  ; HMI IN MOTOR ROLLER3 RVS
@OR 36.02  ; HMI IN MOTOR ROLLER2 FWD
@OR 36.03  ; HMI IN MOTOR ROLLER2 RVS
@OR 36.04  ; HMI IN MOTOR ROLLER1 FWD
@OR 36.05  ; HMI IN MOTOR ROLLER1 RVS
@OR 40.03  ; HMI IN MOTOR ROLLER 5 FWD
@OR 40.04  ; HMI IN MOTOR ROLLER5 RVS
@OR 32.09  ; HMI IN STP1 DN
@OR 32.10  ; HMI IN STP2 UP
@OR 32.11  ; HMI IN STP2 DN
@OR 32.12  ; HMI IN STP3 UP
@OR 32.13  ; HMI IN STP3 DN
@OR 32.14  ; HMI IN STP4 UP
@OR 32.15  ; HMI IN STP4 DN
@OR 33.00  ; HMI IN STP5 UP
@OR 33.01  ; HMI IN STP5 DN
@OR 33.02  ; HMI IN STP6 UP
@OR 33.03  ; HMI IN STP6 DN
@OR 33.04  ; HMI IN STP7 UP
@OR 33.05  ; HMI IN STP7 DN
@OR 33.06  ; HMI IN STP8 UP
@OR 33.07  ; HMI IN STP8 DN
@OR 33.08  ; HMI IN STP9 UP
@OR 33.09  ; HMI IN STP9 DN
@OR 33.10  ; HMI IN STP10 UP
@OR 33.11  ; HMI IN STP10 DN
@OR 33.12  ; HMI IN STP11 UP
@OR 33.13  ; HMI IN STP11 DN
@OR 33.14  ; HMI IN STP12 UP
@OR 33.15  ; HMI IN STP12 DN
@OR 34.00  ; HMI IN STP13 UP
@OR 32.08  ; HMI IN STP1 UP
@OR 34.02  ; HMI IN STP14 UP
@OR 34.01  ; HMI IN STP13 DN
@OR 36.14  ; HMI IN PINLOCK ROT4 UP
@OR 36.15  ; HMI IN PINLOCK ROT4 DN
@OR 37.00  ; HMI IN PINLOCK ROT3 UP
@OR 37.01  ; HMI IN PINLOCK ROT3 DN
@OR 37.02  ; HMI IN PINLOCK ROT2 UP
@OR 37.03  ; HMI IN PIN LOCK ROT2 DN
@OR 37.04  ; HMI IN PINLOCK ROT1 UP
@OR 37.05  ; HMI IIN PIN LOCK ROT1 DN
@OR 34.03  ; HMI IN STP14 DN
@OR 39.03  ; PB HMI HOME POST
@OR 90.02  ; PB HMI RVS ALL
OUT TR0
@ANDNOT 30.00  ; HMI IN M1 FWD
RSET 30.00  ; HMI IN M1 FWD
LD TR0
@ANDNOT 30.01  ; HMI IN M1 RVS
RSET 30.01  ; HMI IN M1 RVS
LD TR0
@ANDNOT 30.02  ; HMI IN M2 FWD
RSET 30.02  ; HMI IN M2 FWD
LD TR0
@ANDNOT 30.03  ; HMI IN M2 RVS
RSET 30.03  ; HMI IN M2 RVS
LD TR0
@ANDNOT 30.04  ; HMI IN M3 FWD
RSET 30.04  ; HMI IN M3 FWD
LD TR0
@ANDNOT 30.05  ; HMI IN M3 RVS
RSET 30.05  ; HMI IN M3 RVS
LD TR0
@ANDNOT 30.06  ; HMI IN M4 FWD
RSET 30.06  ; HMI IN M4 FWD
LD TR0
@ANDNOT 30.07  ; HMI IN M4 RVS
RSET 30.07  ; HMI IN M4 RVS
LD TR0
@ANDNOT 30.08  ; HMI IN M5 FWD
RSET 30.08  ; HMI IN M5 FWD
LD TR0
@ANDNOT 30.09  ; HMI IN M5 RVS
RSET 30.09  ; HMI IN M5 RVS
LD TR0
@ANDNOT 30.10  ; HMI IN M6 FWD
RSET 30.10  ; HMI IN M6 FWD
LD TR0
@ANDNOT 30.11  ; HMI IN M6 RVS
RSET 30.11  ; HMI IN M6 RVS
LD TR0
@ANDNOT 30.12  ; HMI IN M7 FWD
RSET 30.12  ; HMI IN M7 FWD
LD TR0
@ANDNOT 30.13  ; HMI IN M7 RVS
RSET 30.13  ; HMI IN M7 RVS
LD TR0
@ANDNOT 30.14  ; HMI IN M8 FWD
RSET 30.14  ; HMI IN M8 FWD
LD TR0
@ANDNOT 30.15  ; HMI IN M8 RVS
RSET 30.15  ; HMI IN M8 RVS
LD TR0
@ANDNOT 31.00  ; HMI IN M9 FWD
RSET 31.00  ; HMI IN M9 FWD
LD TR0
@ANDNOT 31.01  ; HMI IN M9 RVS
RSET 31.01  ; HMI IN M9 RVS
LD TR0
@ANDNOT 31.02  ; HMI IN M10 FWD
RSET 31.02  ; HMI IN M10 FWD
LD TR0
@ANDNOT 31.03  ; HMI IN M10 RVS
RSET 31.03  ; HMI IN M10 RVS
LD TR0
@ANDNOT 35.14  ; HMI IN MOTOR ROLLER4 FWD
RSET 35.14  ; HMI IN MOTOR ROLLER4 FWD
LD TR0
@ANDNOT 35.15  ; HMI IN MOTOR ROLLER4 RVS
RSET 35.15  ; HMI IN MOTOR ROLLER4 RVS
LD TR0
@ANDNOT 36.00  ; HMI IN MOTOR ROLLER3 FWD
RSET 36.00  ; HMI IN MOTOR ROLLER3 FWD
LD TR0
@ANDNOT 36.01  ; HMI IN MOTOR ROLLER3 RVS
RSET 36.01  ; HMI IN MOTOR ROLLER3 RVS
LD TR0
@ANDNOT 36.02  ; HMI IN MOTOR ROLLER2 FWD
RSET 36.02  ; HMI IN MOTOR ROLLER2 FWD
LD TR0
@ANDNOT 36.03  ; HMI IN MOTOR ROLLER2 RVS
RSET 36.03  ; HMI IN MOTOR ROLLER2 RVS
LD TR0
@ANDNOT 36.04  ; HMI IN MOTOR ROLLER1 FWD
RSET 36.04  ; HMI IN MOTOR ROLLER1 FWD
LD TR0
@ANDNOT 36.05  ; HMI IN MOTOR ROLLER1 RVS
RSET 36.05  ; HMI IN MOTOR ROLLER1 RVS
LD TR0
@ANDNOT 40.03  ; HMI IN MOTOR ROLLER 5 FWD
RSET 40.03  ; HMI IN MOTOR ROLLER 5 FWD
LD TR0
@ANDNOT 40.04  ; HMI IN MOTOR ROLLER5 RVS
RSET 40.04  ; HMI IN MOTOR ROLLER5 RVS
LD TR0
@ANDNOT 32.09  ; HMI IN STP1 DN
RSET 32.09  ; HMI IN STP1 DN
LD TR0
@ANDNOT 32.10  ; HMI IN STP2 UP
RSET 32.10  ; HMI IN STP2 UP
LD TR0
@ANDNOT 32.11  ; HMI IN STP2 DN
RSET 32.11  ; HMI IN STP2 DN
LD TR0
@ANDNOT 32.12  ; HMI IN STP3 UP
RSET 32.12  ; HMI IN STP3 UP
LD TR0
@ANDNOT 32.13  ; HMI IN STP3 DN
RSET 32.13  ; HMI IN STP3 DN
LD TR0
@ANDNOT 32.14  ; HMI IN STP4 UP
RSET 32.14  ; HMI IN STP4 UP
LD TR0
@ANDNOT 32.15  ; HMI IN STP4 DN
RSET 32.15  ; HMI IN STP4 DN
LD TR0
@ANDNOT 33.00  ; HMI IN STP5 UP
RSET 33.00  ; HMI IN STP5 UP
LD TR0
@ANDNOT 33.01  ; HMI IN STP5 DN
RSET 33.01  ; HMI IN STP5 DN
LD TR0
@ANDNOT 33.02  ; HMI IN STP6 UP
RSET 33.02  ; HMI IN STP6 UP
LD TR0
@ANDNOT 33.03  ; HMI IN STP6 DN
RSET 33.03  ; HMI IN STP6 DN
LD TR0
@ANDNOT 33.04  ; HMI IN STP7 UP
RSET 33.04  ; HMI IN STP7 UP
LD TR0
@ANDNOT 33.05  ; HMI IN STP7 DN
RSET 33.05  ; HMI IN STP7 DN
LD TR0
@ANDNOT 33.06  ; HMI IN STP8 UP
RSET 33.06  ; HMI IN STP8 UP
LD TR0
@ANDNOT 33.07  ; HMI IN STP8 DN
RSET 33.07  ; HMI IN STP8 DN
LD TR0
@ANDNOT 33.08  ; HMI IN STP9 UP
RSET 33.08  ; HMI IN STP9 UP
LD TR0
@ANDNOT 33.09  ; HMI IN STP9 DN
RSET 33.09  ; HMI IN STP9 DN
LD TR0
@ANDNOT 33.10  ; HMI IN STP10 UP
RSET 33.10  ; HMI IN STP10 UP
LD TR0
@ANDNOT 33.11  ; HMI IN STP10 DN
RSET 33.11  ; HMI IN STP10 DN
LD TR0
@ANDNOT 33.12  ; HMI IN STP11 UP
RSET 33.12  ; HMI IN STP11 UP
LD TR0
@ANDNOT 33.13  ; HMI IN STP11 DN
RSET 33.13  ; HMI IN STP11 DN
LD TR0
@ANDNOT 33.14  ; HMI IN STP12 UP
RSET 33.14  ; HMI IN STP12 UP
LD TR0
@ANDNOT 33.15  ; HMI IN STP12 DN
RSET 33.15  ; HMI IN STP12 DN
LD TR0
@ANDNOT 34.00  ; HMI IN STP13 UP
RSET 34.00  ; HMI IN STP13 UP
LD TR0
@ANDNOT 32.08  ; HMI IN STP1 UP
RSET 32.08  ; HMI IN STP1 UP
LD TR0
@ANDNOT 34.02  ; HMI IN STP14 UP
RSET 34.02  ; HMI IN STP14 UP
LD TR0
@ANDNOT 34.01  ; HMI IN STP13 DN
RSET 34.01  ; HMI IN STP13 DN
LD TR0
@ANDNOT 36.14  ; HMI IN PINLOCK ROT4 UP
RSET 36.14  ; HMI IN PINLOCK ROT4 UP
LD TR0
@ANDNOT 36.15  ; HMI IN PINLOCK ROT4 DN
RSET 36.15  ; HMI IN PINLOCK ROT4 DN
LD TR0
@ANDNOT 37.00  ; HMI IN PINLOCK ROT3 UP
RSET 37.00  ; HMI IN PINLOCK ROT3 UP
LD TR0
@ANDNOT 37.01  ; HMI IN PINLOCK ROT3 DN
RSET 37.01  ; HMI IN PINLOCK ROT3 DN
LD TR0
@ANDNOT 37.02  ; HMI IN PINLOCK ROT2 UP
RSET 37.02  ; HMI IN PINLOCK ROT2 UP
LD TR0
@ANDNOT 37.03  ; HMI IN PIN LOCK ROT2 DN
RSET 37.03  ; HMI IN PIN LOCK ROT2 DN
LD TR0
@ANDNOT 37.04  ; HMI IN PINLOCK ROT1 UP
RSET 37.04  ; HMI IN PINLOCK ROT1 UP
LD TR0
@ANDNOT 37.05  ; HMI IIN PIN LOCK ROT1 DN
RSET 37.05  ; HMI IIN PIN LOCK ROT1 DN
LD TR0
@ANDNOT 34.03  ; HMI IN STP14 DN
RSET 34.03  ; HMI IN STP14 DN
LD TR0
@ANDNOT 39.03  ; PB HMI HOME POST
RSET 39.03  ; PB HMI HOME POST
LD TR0
@ANDNOT 90.02  ; PB HMI RVS ALL
RSET 90.02  ; PB HMI RVS ALL

